// TwinCAT 3 PLC project MobilePlatform
// ProgramVersion: 3.1.4022.7
// libraries:
//   Tc2_EtherCAT, * (Beckhoff Automation GmbH)
//   Tc2_Math, * (Beckhoff Automation GmbH)
//   Tc2_MC2, * (Beckhoff Automation GmbH)
//   Tc2_Standard, * (Beckhoff Automation GmbH)
//   Tc2_SUPS, * (Beckhoff Automation GmbH)
//   Tc2_System, * (Beckhoff Automation GmbH)
//   Tc2_TcpIp, * (Beckhoff Automation GmbH)
//   Tc2_Utilities, * (Beckhoff Automation GmbH)
//   Tc3_Module, * (Beckhoff Automation GmbH)
// project tree:
//   DUTs/ ButtonType.TcDUT, ByteDword.TcDUT, ByteReal.TcDUT, ControlerState.TcDUT, DirPlatform.TcDUT, E_ClientServerSteps.TcDUT, E_CONTROL_STATES.TcDUT, InternalState.TcDUT, JoystickCalibState.TcDUT, JoystickState.TcDUT, LEDtype.TcDUT, RealDword.TcDUT, ST_Calibration_Parameters.TcDUT, ST_FrameFifoEntry.TcDUT
//   GVLs/ ControlGVL.TcGVL, JoystickGVL.TcGVL, MOTORS.TcGVL, SafetyGVL.TcGVL, SensorsGVL.TcGVL
//   POUs/Joystick/FBs/ AXISdriver.TcPOU, BUTTONdriver.TcPOU, CalibrationFB.TcPOU, LEDdriver.TcPOU
//   POUs/Joystick/ JoystickMain.TcPOU
//   POUs/Motors/FBs/ FB_RESET_MOTORS.TcPOU, FB_RUN_MOTOR.TcPOU
//   POUs/Motors/ MAIN.TcPOU
//   POUs/Sensors/ SensorsMain.TcPOU
//   / Task1.TcTTO, Task3.TcTTO, Task_2.TcTTO
// real-time tasks:
//   TASK Task1: cycle T#50us, priority 6, ADS port 350
//   TASK Task3: cycle T#10ms, priority 12, ADS port 360
//   TASK Task 2: cycle T#1ms, priority 7, ADS port 351
// motion (NC):
//   TASK NC-Task 1 SAF: cycle T#500us, priority 8, ADS port 501
//   TASK NC-Task 1 SVB: cycle T#10ms, priority 14, ADS port 511
//   AXIS Wheel_Back_Left (id 1)
//     General: UnitName=°
//     Dynamic: Acceleration=30537, Deceleration=30537, Jerk=91611
//     Velo: RefSearch=203.58, RefSync=203.58, SlowManual=1017.9, FastManual=6107.4, Fast=20358, Maximum=20358
//     OtherSettings: AllowMotionCmdToSlave=true
//     encoder EncType=19
//       EncPara: ScaleFactorNumerator=360, ScaleFactorDenominator=1048576, MaxCount=#xffffffff
//     drive DrvType=16
//       DrvPara: MaxCount=#xffffffff, DriveControlDWord=#x00020000
//         Analog: VeloReferenz=22393.8, VeloScale=32, ScaleFactorActTorque=0.1
//         TimeComp: TaskDelayCycles=1
//     controller CtrType=1
//       CtrPara: PriorControlFactor=1
//         PosDiffControl: Enable=false
//         Observer: BandWidth=20
//   AXIS Wheel_Back_Right (id 2)
//     General: UnitName=°
//     Dynamic: Acceleration=30537, Deceleration=30537, Jerk=91611
//     Velo: RefSearch=203.58, RefSync=203.58, SlowManual=1017.9, FastManual=6107.4, Fast=20358, Maximum=20358
//     OtherSettings: AllowMotionCmdToSlave=true
//     encoder EncType=19
//       EncPara: ScaleFactorNumerator=360, ScaleFactorDenominator=1048576, MaxCount=#xffffffff
//     drive DrvType=16
//       DrvPara: MaxCount=#xffffffff, DriveControlDWord=#x00020000
//         Analog: VeloReferenz=22393.8, VeloScale=32, ScaleFactorActTorque=0.1
//         TimeComp: TaskDelayCycles=1
//     controller CtrType=1
//       CtrPara: PriorControlFactor=1
//         PosDiffControl: Enable=false
//         Observer: BandWidth=20
//   AXIS Wheel_Front_Left (id 3)
//     General: UnitName=°
//     Dynamic: Acceleration=30537, Deceleration=30537, Jerk=91611
//     Velo: RefSearch=203.58, RefSync=203.58, SlowManual=1017.9, FastManual=6107.4, Fast=20358, Maximum=20358
//     OtherSettings: AllowMotionCmdToSlave=true
//     encoder EncType=19
//       EncPara: ScaleFactorNumerator=360, ScaleFactorDenominator=1048576, MaxCount=#xffffffff
//     drive DrvType=16
//       DrvPara: MaxCount=#xffffffff, DriveControlDWord=#x00020000
//         Analog: VeloReferenz=22393.8, VeloScale=32, ScaleFactorActTorque=0.1
//         TimeComp: TaskDelayCycles=1
//     controller CtrType=1
//       CtrPara: PriorControlFactor=1
//         PosDiffControl: Enable=false
//         Observer: BandWidth=20
//   AXIS Wheel_Front_Right (id 4)
//     General: UnitName=°
//     Dynamic: Acceleration=30537, Deceleration=30537, Jerk=91611
//     Velo: RefSearch=203.58, RefSync=203.58, SlowManual=1017.9, FastManual=6107.4, Fast=20358, Maximum=20358
//     OtherSettings: AllowMotionCmdToSlave=true
//     encoder EncType=19
//       EncPara: ScaleFactorNumerator=360, ScaleFactorDenominator=1048576, MaxCount=#xffffffff
//     drive DrvType=16
//       DrvPara: MaxCount=#xffffffff, DriveControlDWord=#x00020000
//         Analog: VeloReferenz=22393.8, VeloScale=32, ScaleFactorActTorque=0.1
//         TimeComp: TaskDelayCycles=1
//     controller CtrType=1
//       CtrPara: PriorControlFactor=1
//         PosDiffControl: Enable=false
//         Observer: BandWidth=20
// I/O:
//   DEVICE Device 1 (EtherCAT), AmsNetId 5.51.149.114.2.1
//     Term 1 (EK1200) [EK1200-5000 EtherCAT Power supply (2A E-Bus)]
//       Term 2 (EL3008) [EL3008 8Ch. Ana. Input +/-10V]
//       Term 3 (EL1259) [EL1259 8Ch. Dig Input 24V/8Ch. Dig. Output 24V with Multi-Time-Stamp]
//       Term 4 (EL7211-9014) [EL7211-9014 1Ch. MDP742 Servo motor output stage with OCT (50V, 4.5A RMS) and STO input]
//       Term 5 (EL7211-9014) [EL7211-9014 1Ch. MDP742 Servo motor output stage with OCT (50V, 4.5A RMS) and STO input]
//       Term 6 (EL2904) [EL2904, 4 Ch. Safety Output 24V, 0.5A, TwinSAFE]
//         modules: Module 1 (FSOES), Module 2 (DO)
//       Term 7 (EL7211-9014) [EL7211-9014 1Ch. MDP742 Servo motor output stage with OCT (50V, 4.5A RMS) and STO input]
//       Term 8 (EL7211-9014) [EL7211-9014 1Ch. MDP742 Servo motor output stage with OCT (50V, 4.5A RMS) and STO input]
//       Term 9 (EL1904) [EL1904, 4 Ch. Safety Input 24V, TwinSAFE]
//         modules: Module 1 (FSOES)
//       Term 10 (EL6900) [EL6900, TwinSAFE PLC]
//       Term 11 (EL6070) [EL6070 1Ch. Licensing-Terminal]
//       Term 12 (EL9011) [EL9011 End Terminal]
// variable links:
//   Device 1 (EtherCAT) <-> Device 1 (EtherCAT)/Term 1 (EK1200)/Term 10 (EL6900)
//     Term 1 (EK1200)/Term 6 (EL2904)/Module 1 (FSOES)/RxPDO/FSOE <-> ConnectionInputs/Message_2 TxPDO
//     Term 1 (EK1200)/Term 9 (EL1904)/Module 1 (FSOES)/RxPDO/FSOE <-> ConnectionInputs/Message_3 TxPDO
//   Device 1 (EtherCAT) <-> Device 1 (EtherCAT)/Term 1 (EK1200)/Term 6 (EL2904)
//     Term 1 (EK1200)/Term 10 (EL6900)/ConnectionOutputs/Message_2 RxPDO <-> Module 1 (FSOES)/TxPDO/FSOE
//   Device 1 (EtherCAT) <-> Device 1 (EtherCAT)/Term 1 (EK1200)/Term 9 (EL1904)
//     Term 1 (EK1200)/Term 10 (EL6900)/ConnectionOutputs/Message_3 RxPDO <-> Module 1 (FSOES)/TxPDO/FSOE
//   NC-Task 1 SAF/Axes/Wheel_Back_Left <-> Device 1 (EtherCAT)/Term 1 (EK1200)/Term 4 (EL7211-9014)
//     Drive/Inputs/In/nDcOutputTime <-> InfoData/DcOutputShift
//     Drive/Inputs/In/nState1 <-> DRV Statusword/Statusword
//     Drive/Inputs/In/nState2 <-> DRV Statusword/Statusword @bit 8
//     Drive/Inputs/In/nState4 @bit 1 <-> WcState/InputToggle
//     Drive/Inputs/In/nState4 <-> WcState/WcState
//     Drive/Outputs/Out/nCtrl1 <-> DRV Controlword/Controlword
//     Drive/Outputs/Out/nCtrl2 <-> DRV Controlword/Controlword @bit 8
//     Drive/Outputs/Out/nDataOut2 <-> DRV Target velocity/Target velocity
//     Enc/Inputs/In/nDataIn1 <-> FB Position/Position
//     Enc/Inputs/In/nDcInputTime <-> InfoData/DcInputShift
//     Enc/Inputs/In/nState4 @bit 1 <-> WcState/InputToggle
//     Enc/Inputs/In/nState4 <-> WcState/WcState
//   NC-Task 1 SAF/Axes/Wheel_Back_Right <-> Device 1 (EtherCAT)/Term 1 (EK1200)/Term 5 (EL7211-9014)
//     Drive/Inputs/In/nDcOutputTime <-> InfoData/DcOutputShift
//     Drive/Inputs/In/nState1 <-> DRV Statusword/Statusword
//     Drive/Inputs/In/nState2 <-> DRV Statusword/Statusword @bit 8
//     Drive/Inputs/In/nState4 @bit 1 <-> WcState/InputToggle
//     Drive/Inputs/In/nState4 <-> WcState/WcState
//     Drive/Outputs/Out/nCtrl1 <-> DRV Controlword/Controlword
//     Drive/Outputs/Out/nCtrl2 <-> DRV Controlword/Controlword @bit 8
//     Drive/Outputs/Out/nDataOut2 <-> DRV Target velocity/Target velocity
//     Enc/Inputs/In/nDataIn1 <-> FB Position/Position
//     Enc/Inputs/In/nDcInputTime <-> InfoData/DcInputShift
//     Enc/Inputs/In/nState4 @bit 1 <-> WcState/InputToggle
//     Enc/Inputs/In/nState4 <-> WcState/WcState
//   NC-Task 1 SAF/Axes/Wheel_Front_Left <-> Device 1 (EtherCAT)/Term 1 (EK1200)/Term 7 (EL7211-9014)
//     Drive/Inputs/In/nDcOutputTime <-> InfoData/DcOutputShift
//     Drive/Inputs/In/nState1 <-> DRV Statusword/Statusword
//     Drive/Inputs/In/nState2 <-> DRV Statusword/Statusword @bit 8
//     Drive/Inputs/In/nState4 @bit 1 <-> WcState/InputToggle
//     Drive/Inputs/In/nState4 <-> WcState/WcState
//     Drive/Outputs/Out/nCtrl1 <-> DRV Controlword/Controlword
//     Drive/Outputs/Out/nCtrl2 <-> DRV Controlword/Controlword @bit 8
//     Drive/Outputs/Out/nDataOut2 <-> DRV Target velocity/Target velocity
//     Enc/Inputs/In/nDataIn1 <-> FB Position/Position
//     Enc/Inputs/In/nDcInputTime <-> InfoData/DcInputShift
//     Enc/Inputs/In/nState4 @bit 1 <-> WcState/InputToggle
//     Enc/Inputs/In/nState4 <-> WcState/WcState
//   NC-Task 1 SAF/Axes/Wheel_Front_Right <-> Device 1 (EtherCAT)/Term 1 (EK1200)/Term 8 (EL7211-9014)
//     Drive/Inputs/In/nDcOutputTime <-> InfoData/DcOutputShift
//     Drive/Inputs/In/nState1 <-> DRV Statusword/Statusword
//     Drive/Inputs/In/nState2 <-> DRV Statusword/Statusword @bit 8
//     Drive/Inputs/In/nState4 @bit 1 <-> WcState/InputToggle
//     Drive/Inputs/In/nState4 <-> WcState/WcState
//     Drive/Outputs/Out/nCtrl1 <-> DRV Controlword/Controlword
//     Drive/Outputs/Out/nCtrl2 <-> DRV Controlword/Controlword @bit 8
//     Drive/Outputs/Out/nDataOut2 <-> DRV Target velocity/Target velocity
//     Enc/Inputs/In/nDataIn1 <-> FB Position/Position
//     Enc/Inputs/In/nDcInputTime <-> InfoData/DcInputShift
//     Enc/Inputs/In/nState4 @bit 1 <-> WcState/InputToggle
//     Enc/Inputs/In/nState4 <-> WcState/WcState
//   MobilePlatform/MobilePlatform Instance <-> Device 1 (EtherCAT)/Term 1 (EK1200)/Term 10 (EL6900)
//     Task1 Inputs/SafetyGVL.ComErr <-> StandardInputs/Standard Out Var 4
//     Task1 Inputs/SafetyGVL.EStop <-> StandardInputs/Standard Out Var 5
//     Task1 Outputs/SafetyGVL.ErrAck <-> StandardOutputs/Standard In Var 1
//   MobilePlatform/MobilePlatform Instance <-> Device 1 (EtherCAT)/Term 1 (EK1200)/Term 2 (EL3008)
//     Task3 Inputs/JoystickMain.axDr.xRaw <-> AI Standard Channel 1/Value
//     Task3 Inputs/JoystickMain.axDr.yRaw <-> AI Standard Channel 2/Value
//     Task3 Inputs/JoystickMain.axDr.zRaw <-> AI Standard Channel 3/Value
//     Task3 Inputs/JoystickMain.calFB.axDr.xRaw <-> AI Standard Channel 1/Value
//     Task3 Inputs/JoystickMain.calFB.axDr.yRaw <-> AI Standard Channel 2/Value
//     Task3 Inputs/JoystickMain.calFB.axDr.zRaw <-> AI Standard Channel 3/Value
//   MobilePlatform/MobilePlatform Instance <-> Device 1 (EtherCAT)/Term 1 (EK1200)/Term 3 (EL1259)
//     Task3 Inputs/JoystickMain.btDR.ch1 <-> MTI Inputs 10x Channel 1/Status/Input state
//     Task3 Inputs/JoystickMain.btDR.ch8 <-> MTI Inputs 10x Channel 8/Status/Input state
//     Task3 Outputs/JoystickMain.ldDr1.ch1 <-> MTO Outputs 10x Channel 1/Ctrl/Manual output state
//     Task3 Outputs/JoystickMain.ldDr3.ch3 <-> MTO Outputs 10x Channel 3/Ctrl/Manual output state
//     Task3 Outputs/JoystickMain.ldDr1.ch1mode <-> MTO Outputs 10x Channel 1/Ctrl/Enable manual operation
//     Task3 Outputs/JoystickMain.ldDr3.ch3mode <-> MTO Outputs 10x Channel 3/Ctrl/Enable manual operation
//     Task_2 Inputs/SensorsMain.sensor1_UO1 <-> MTI Inputs 10x Channel 5/Status/Input state
//     Task_2 Inputs/SensorsMain.sensor1_UO2 <-> MTI Inputs 10x Channel 6/Status/Input state
//     Task_2 Inputs/SensorsMain.sensor1_UO3 <-> MTI Inputs 10x Channel 4/Status/Input state
//     Task_2 Inputs/SensorsMain.sensor2_UO1 <-> MTI Inputs 10x Channel 2/Status/Input state
//     Task_2 Inputs/SensorsMain.sensor2_UO2 <-> MTI Inputs 10x Channel 3/Status/Input state
//     Task_2 Inputs/SensorsMain.sensor2_UO3 <-> MTI Inputs 10x Channel 7/Status/Input state
//     Task_2 Outputs/SensorsMain.en_sensor1_D <-> MTO Outputs 10x Channel 6/Ctrl/Enable manual operation
//     Task_2 Outputs/SensorsMain.en_sensor2_D <-> MTO Outputs 10x Channel 5/Ctrl/Enable manual operation
//     Task_2 Outputs/SensorsMain.en_sensor1_E <-> MTO Outputs 10x Channel 7/Ctrl/Enable manual operation
//     Task_2 Outputs/SensorsMain.en_sensor2_E <-> MTO Outputs 10x Channel 4/Ctrl/Enable manual operation
//     Task_2 Outputs/SensorsMain.en_sensor1_F <-> MTO Outputs 10x Channel 8/Ctrl/Enable manual operation
//     Task_2 Outputs/SensorsMain.en_sensor2_F <-> MTO Outputs 10x Channel 2/Ctrl/Enable manual operation
//     Task_2 Outputs/SensorsMain.sensor1_D <-> MTO Outputs 10x Channel 6/Ctrl/Manual output state
//     Task_2 Outputs/SensorsMain.sensor2_D <-> MTO Outputs 10x Channel 5/Ctrl/Manual output state
//     Task_2 Outputs/SensorsMain.sensor1_E <-> MTO Outputs 10x Channel 7/Ctrl/Manual output state
//     Task_2 Outputs/SensorsMain.sensor2_E <-> MTO Outputs 10x Channel 4/Ctrl/Manual output state
//     Task_2 Outputs/SensorsMain.sensor1_F <-> MTO Outputs 10x Channel 8/Ctrl/Manual output state
//     Task_2 Outputs/SensorsMain.sensor2_F <-> MTO Outputs 10x Channel 2/Ctrl/Manual output state
//   MobilePlatform/MobilePlatform Instance <-> NC-Task 1 SAF/Axes/Wheel_Back_Left
//     Task1 Inputs/MOTORS.fbAxisRef_BL.NcToPlc <-> Outputs/ToPlc
//     Task1 Outputs/MOTORS.fbAxisRef_BL.PlcToNc <-> Inputs/FromPlc
//   MobilePlatform/MobilePlatform Instance <-> NC-Task 1 SAF/Axes/Wheel_Back_Right
//     Task1 Inputs/MOTORS.fbAxisRef_BR.NcToPlc <-> Outputs/ToPlc
//     Task1 Outputs/MOTORS.fbAxisRef_BR.PlcToNc <-> Inputs/FromPlc
//   MobilePlatform/MobilePlatform Instance <-> NC-Task 1 SAF/Axes/Wheel_Front_Left
//     Task1 Inputs/MOTORS.fbAxisRef_FL.NcToPlc <-> Outputs/ToPlc
//     Task1 Outputs/MOTORS.fbAxisRef_FL.PlcToNc <-> Inputs/FromPlc
//   MobilePlatform/MobilePlatform Instance <-> NC-Task 1 SAF/Axes/Wheel_Front_Right
//     Task1 Inputs/MOTORS.fbAxisRef_FR.NcToPlc <-> Outputs/ToPlc
//     Task1 Outputs/MOTORS.fbAxisRef_FR.PlcToNc <-> Inputs/FromPlc

CONFIGURATION MobilePlatform
    RESOURCE PLC ON TwinCAT3
        TASK Task1(INTERVAL := T#50us, PRIORITY := 6);
        TASK Task3(INTERVAL := T#10ms, PRIORITY := 12);
        TASK Task_2(INTERVAL := T#1ms, PRIORITY := 7);
        PROGRAM MAIN WITH Task1 : MAIN;
        PROGRAM JoystickMain WITH Task3 : JoystickMain;
        PROGRAM SensorsMain WITH Task_2 : SensorsMain;
    END_RESOURCE
END_CONFIGURATION

// ---- DUTs/ButtonType.TcDUT
{attribute 'qualified_only'}
//{attribute 'strict'}
TYPE ButtonType :
(
	notPressed := 0,
	pressed := 1,
	hold2s := 2,
	hold5s := 5
);
END_TYPE

// ---- DUTs/ByteDword.TcDUT
TYPE ByteDword :
UNION
	dValue : DWORD;    // Needs 4 Bytes in memory
    abValue:  ARRAY [1..4] OF BYTE;
END_UNION
END_TYPE

// ---- DUTs/ByteReal.TcDUT
TYPE ByteReal :
UNION
	rValue : REAL;    // Needs 4 Bytes in memory
    abValue:  ARRAY [1..4] OF BYTE;
END_UNION
END_TYPE

// ---- DUTs/ControlerState.TcDUT
{attribute 'qualified_only'}
{attribute 'strict'}
TYPE ControlerState :
(
	UDPcontrol := 0,
	LocalOverride := 1,
	Blocked := 2
);
END_TYPE

// ---- DUTs/DirPlatform.TcDUT
{attribute 'qualified_only'}
{attribute 'strict'}
TYPE DirPlatform :
(
	
	PLUS_X := 0,
	PLUS_X_MINUS_Y := 1,
	MINUS_Y := 2,
	MINUS_X_MINUS_Y := 3,
	MINUS_X := 4,
	MINUS_X_PLUS_Y := 5,
	PLUS_Y := 6,
	PLUS_X_PLUS_Y := 7
);
END_TYPE

// ---- DUTs/E_ClientServerSteps.TcDUT
TYPE E_ClientServerSteps :
(
	eUDP_STATE_IDLE		:= 0,
	eUDP_STATE_CREATE_START,
	eUDP_STATE_CREATE_WAIT,
	eUDP_STATE_SEND_START,
	eUDP_STATE_SEND_WAIT,
	eUDP_STATE_RECEIVE_START,
	eUDP_STATE_RECEIVE_WAIT,
	eUDP_STATE_CLOSE_START,
	eUDP_STATE_CLOSE_WAIT,
	eUDP_STATE_ERROR
);
END_TYPE

// ---- DUTs/E_CONTROL_STATES.TcDUT
TYPE E_CONTROL_STATES :
(
	eControlState_Preinit := 100,
	eControlState_Init := 110,
	eControlState_Hold := 120,
	eControlState_Move := 130,
	eControlState_Move_Omni := 140,
	eControlState_Move_Omni_Rot := 150
	);
END_TYPE

// ---- DUTs/InternalState.TcDUT
{attribute 'qualified_only'}
{attribute 'strict'}
TYPE InternalState :
(
	passive := 0,
	override := 1,
	udpOnly := 2
);
END_TYPE

// ---- DUTs/JoystickCalibState.TcDUT
{attribute 'qualified_only'}
{attribute 'strict'}
TYPE JoystickCalibState :
(
	CalibMinMax := 0,
	CalibDeadband := 1,
	CalibOver := 2,
	CalibStart := 3
);
END_TYPE

// ---- DUTs/JoystickState.TcDUT
{attribute 'qualified_only'}
{attribute 'strict'}
TYPE JoystickState :
(
	NoCalib := 0,
	Operational := 1,
	Calib := 2
);
END_TYPE

// ---- DUTs/LEDtype.TcDUT
{attribute 'qualified_only'}
{attribute 'strict'}
TYPE LEDtype :
(
	OFF := 0,
	ON := 1,
	Pulse := 2,
	BlinkOnce := 3,
	BlinkContinious := 4
);
END_TYPE

// ---- DUTs/RealDword.TcDUT
TYPE RealDword :
UNION
	rValue : REAL;
	dValue : DWORD;
END_UNION
END_TYPE

// ---- DUTs/ST_Calibration_Parameters.TcDUT
TYPE ST_Calibration_Parameters :
STRUCT
	maximums : ARRAY [1..3] OF INT;
	minimums : ARRAY [1..3] OF INT;
	deadband : ARRAY [1..3] OF INT;
	zero     : ARRAY [1..3] OF INT;
	
	timeOfCalib : DATE_AND_TIME;
	
	calibrated : BOOL := FALSE;
END_STRUCT
END_TYPE

// ---- DUTs/ST_FrameFifoEntry.TcDUT
TYPE ST_FrameFifoEntry :
STRUCT
	stRemoteAddr 	: ST_SockAddr;(* Remote address. String containing an (Ipv4) Internet Protocol dotted address and port number. *)
	sMessage		: ARRAY [0..100] OF BYTE;	(* UDP packet data *)
END_STRUCT
END_TYPE

// ---- GVLs/ControlGVL.TcGVL
{attribute 'qualified_only'}
VAR_GLOBAL


	
	status : DWORD := 0; //status Bit0 - EStop Active, Bit1 - Manual override, Bit2 - JoystickUdp only, Bit3 - 9 Joystick states
	//all values in deg or deg/s
	vel_BL : LREAL := 0.0;
	vel_BR : LREAL := 0.0;
	vel_FL : LREAL := 0.0;
	vel_FR : LREAL := 0.0;
	
	pos_BL : LREAL := 0.0;
	pos_BR : LREAL := 0.0;
	pos_FL : LREAL := 0.0;
	pos_FR : LREAL := 0.0;
	
	leftRight : LREAL := 0; // left-right command 
	forwardReverse : LREAL := 0; // forward-reverse comand
	rotLeftRight : LREAL := 0;
	
	TimeStamp : LREAL := 0.0;
	
	vel_robot : ARRAY [1..3] OF LREAL := [0,0,0]; //commands platform velocity x-y-th + timestamp	from ROS
	robot_odom : ARRAY [1..6] OF LREAL := [0,0,0,0,0,0]; //acctual position and velocity robot order pos-vel x-y-th
	
	
	currentVelMax : LREAL :=0;
	currentThVelMax : LREAL :=0;
END_VAR

// ---- GVLs/JoystickGVL.TcGVL
{attribute 'qualified_only'}
VAR_GLOBAL
	state : JoystickState := JoystickState.NoCalib;
	xConst : LREAL := -0.3; //x y z max speeds
	yConst : LREAL := 0.2;
	zConst : LREAL := 0.4;
	
	xSpeed : LREAL := 0.0;
	ySpeed : LREAL := 0.0;
	zSpeed : LREAL := 0.0;
	
	speedScale : LREAL := 1.0;
	
	intState : InternalState := InternalState.passive;
	
	lastUpdate : BOOL := FALSE;
	lastExec : BOOL := FALSE;
END_VAR

VAR_GLOBAL PERSISTENT
	calibration : ST_Calibration_Parameters;
END_VAR

// ---- GVLs/MOTORS.TcGVL
{attribute 'qualified_only'}

VAR_GLOBAL
	
    // Axis reference 
    fbAxisRef_BL:				AXIS_REF;
	fbAxisRef_BR:				AXIS_REF;
	fbAxisRef_FL:				AXIS_REF;
	fbAxisRef_FR:				AXIS_REF;
	// Motors' Power
	fbPOWER_BL : 				MC_Power;
    fbPOWER_BR : 				MC_Power;	
    fbPOWER_FL : 				MC_Power;
    fbPOWER_FR : 				MC_Power;		
	// Reset Motors
	fbRESET_BL : 				MC_Reset;
	fbRESET_BR : 				MC_Reset;
	// Stop Motors
	fbSTOP_BL :	 				MC_Stop;
	fbSTOP_BR :	 				MC_Stop;
	// Velocity Controllers 
	fbVELOCITY_BL : 			MC_MoveVelocity;
	fbVELOCITY_BR : 			MC_MoveVelocity;
	fbVELOCITY_FL : 			MC_MoveVelocity;
	fbVELOCITY_FR : 			MC_MoveVelocity;
	// Move absolute - it will move the axis to an absolute position 
	fbMOVEABSOLUTE_LB : 		MC_MoveAbsolute;
	fbMOVEABSOLUTE_RB : 		MC_MoveAbsolute;
	// Set position if mode relative
	fbSETPOSITION_BL : 			MC_SetPosition;
	fbSETPOSITION_BR : 			MC_SetPosition;
    // Move relative - it will move the axis to a relative position
	fbMOVERELATIVE_BL : 		MC_MoveRelative;
	fbMOVERELATIVE_BR : 		MC_MoveRelative;
	// Read actual position of the axis
	fbACTUALPOSITION_BL : 		MC_ReadActualPosition;
	fbACTUALPOSITION_BR : 		MC_ReadActualPosition;
	// Direction enumeration
	fbDirection_BL: 			MC_Direction := MC_Positive_Direction;  // MC_Positive_Direction or MC_Negative_Direction
	fbDirection_BR: 			MC_Direction := MC_Positive_Direction; 
	fbDirection_FL: 			MC_Direction := MC_Positive_Direction;  // MC_Positive_Direction or MC_Negative_Direction
	fbDirection_FR: 			MC_Direction := MC_Positive_Direction; 
	
	// Control Values
	bAxis_Ready : 				BOOL;
	b_Move_Absolut_Aborted : 	BOOL;
	bReset_Done : 				BOOL;
    lrAcc_Axis_1 : 				LREAL;
	lrActual_Position : 		LREAL;
	lrDecel_Axis_1 :			LREAL;
	lrJerk_Axis_1 : 			LREAL;
	lrPosition_Drive_to : 		LREAL;
	lrVelocity_Move_Ab_Axis: 	LREAL;	
	
	//External set point generators enable
	MC_ExtSetPointGenEnableBL : MC_ExtSetPointGenEnable;
	MC_ExtSetPointGenEnableBR : MC_ExtSetPointGenEnable;
	MC_ExtSetPointGenEnableFL : MC_ExtSetPointGenEnable;
	MC_ExtSetPointGenEnableFR : MC_ExtSetPointGenEnable;
	
	//External set point generators disable
	MC_ExtSetPointGenDisableBL : MC_ExtSetPointGenDisable;
	MC_ExtSetPointGenDisableBR : MC_ExtSetPointGenDisable;
	MC_ExtSetPointGenDisableFL : MC_ExtSetPointGenDisable;
	MC_ExtSetPointGenDisableFR : MC_ExtSetPointGenDisable;


	

END_VAR

// ---- GVLs/SafetyGVL.TcGVL
{attribute 'qualified_only'}
VAR_GLOBAL
	ErrAck AT %Q* : BOOL;
	ComErr AT %I* : BOOL;
	EStop AT %I* : BOOL;
END_VAR

// ---- GVLs/SensorsGVL.TcGVL
{attribute 'qualified_only'}
VAR_GLOBAL

	
	platformDir : INT := 0;

END_VAR

// ---- POUs/Motors/MAIN.TcPOU
PROGRAM MAIN
VAR
	

	tmr1 : TON;
	tmr1val : BOOL := FALSE;
	
	estopActive : BOOL := FALSE;
	
	reset1 : FB_RESET_MOTORS;
	
	Enabled : BOOL := TRUE;
	
	fbRunMotor : FB_RUN_MOTOR;
	//leddriver : LEDdriver;
END_VAR

IF SafetyGVL.ComErr = TRUE THEN
	//Safety needs to be reset - reset safety
	SafetyGVL.ErrAck := TRUE;
	tmr1val := TRUE;
END_IF

IF SafetyGVL.EStop = FALSE THEN
		//EStop was activated
		estopActive := TRUE;
		ControlGVL.status := ControlGVL.status OR 2#00000000000000000000000000000001;
END_IF

tmr1(IN := tmr1val, PT := T#1S);

IF (estopActive = TRUE) AND (SafetyGVL.EStop = TRUE) THEN
	//EStop over - reset motor drivers
	reset1();
	IF reset1.EstopOut = FALSE THEN
		ControlGVL.status := ControlGVL.status AND 2#11111111111111111111111111111110;
		estopActive := FALSE;
	END_IF
END_IF

IF tmr1.Q = TRUE THEN
	
	//Safety online - run program
	SafetyGVL.ErrAck := FALSE;
	fbRunMotor();
	//leddriver(ledBlink := LEDtype.ON, blinkInterval := T#1S, ledChannel := 3);
	
END_IF

END_PROGRAM

// ---- POUs/Motors/FBs/FB_RESET_MOTORS.TcPOU
FUNCTION_BLOCK FB_RESET_MOTORS
VAR_INPUT
END_VAR
VAR_OUTPUT
	EstopOut : BOOL := TRUE;
END_VAR
VAR
	tmr1 : TON;
	
	tmr1val : BOOL := FALSE;
	
	reset1 : MC_Reset;
	reset2 : MC_Reset;
	reset3 : MC_Reset;
	reset4 : MC_Reset;
END_VAR

tmr1(IN := tmr1val, PT :=T#2S);

IF tmr1.Q = FALSE THEN
	
	reset1(Axis := MOTORS.fbAxisRef_BL, Execute := TRUE);
	reset2(Axis := MOTORS.fbAxisRef_BR, Execute := TRUE);
	reset3(Axis := MOTORS.fbAxisRef_FR, Execute := TRUE);
	reset4(Axis := MOTORS.fbAxisRef_FL, Execute := TRUE);
	tmr1val := TRUE;
	EstopOut := TRUE;
	
	//disable use of external set point generator
	MOTORS.MC_ExtSetPointGenDisableBL(Axis:=MOTORS.fbAxisRef_BL,
		Execute := TRUE);
	MOTORS.MC_ExtSetPointGenDisableBR(Axis:=MOTORS.fbAxisRef_BR,
		Execute := TRUE);
	MOTORS.MC_ExtSetPointGenDisableFR(Axis:=MOTORS.fbAxisRef_FR,
		Execute := TRUE);
	MOTORS.MC_ExtSetPointGenDisableFL(Axis:=MOTORS.fbAxisRef_FL,
		Execute := TRUE);
			
	//reset enable
	MOTORS.MC_ExtSetPointGenEnableBL(Axis:=MOTORS.fbAxisRef_BL,
		Execute:=FALSE);
	MOTORS.MC_ExtSetPointGenEnableBR(Axis:=MOTORS.fbAxisRef_BR,
		Execute:=FALSE);
	MOTORS.MC_ExtSetPointGenEnableFL(Axis:=MOTORS.fbAxisRef_FL,
		Execute:=FALSE);
	MOTORS.MC_ExtSetPointGenEnableFR(Axis:=MOTORS.fbAxisRef_FR,
		Execute:=FALSE);
	
	
END_IF

IF tmr1.Q = TRUE THEN
	
	reset1(Axis := MOTORS.fbAxisRef_BL, Execute := FALSE);
	reset2(Axis := MOTORS.fbAxisRef_BR, Execute := FALSE);
	reset3(Axis := MOTORS.fbAxisRef_FR, Execute := FALSE);
	reset4(Axis := MOTORS.fbAxisRef_FL, Execute := FALSE);
	tmr1val := FALSE;
	EstopOut := FALSE;
	
	
		
		//Enable use of external set point generator
	MOTORS.MC_ExtSetPointGenEnableBL(Axis:=MOTORS.fbAxisRef_BL,
		Execute:=TRUE,
		Position := 0,
		PositionType:=POSITIONTYPE_ABSOLUTE);
		
	MOTORS.MC_ExtSetPointGenEnableBR(Axis:=MOTORS.fbAxisRef_BR,
		Execute:=TRUE,
		Position := 0,
		PositionType:=POSITIONTYPE_ABSOLUTE);
			
	MOTORS.MC_ExtSetPointGenEnableFL(Axis:=MOTORS.fbAxisRef_FL,
		Execute:=TRUE,
		Position := 0,
		PositionType:=POSITIONTYPE_ABSOLUTE);
			
	MOTORS.MC_ExtSetPointGenEnableFR(Axis:=MOTORS.fbAxisRef_FR,
		Execute:=TRUE,
		Position := 0,
		PositionType:=POSITIONTYPE_ABSOLUTE);
			
	//reset disable external setpoint
	MOTORS.MC_ExtSetPointGenDisableBL(Axis:=MOTORS.fbAxisRef_BL,
		Execute := FALSE);
	MOTORS.MC_ExtSetPointGenDisableBR(Axis:=MOTORS.fbAxisRef_BR,
		Execute := FALSE);	
	MOTORS.MC_ExtSetPointGenDisableFR(Axis:=MOTORS.fbAxisRef_FR,
		Execute := FALSE);	
	MOTORS.MC_ExtSetPointGenDisableFL(Axis:=MOTORS.fbAxisRef_FL,
		Execute := FALSE);
END_IF

END_FUNCTION_BLOCK

// ---- POUs/Motors/FBs/FB_RUN_MOTOR.TcPOU
FUNCTION_BLOCK FB_RUN_MOTOR

VAR
	fbTMR : TON;
    Count : INT := 0;
    
    EnableMoveMotor : BOOL := FALSE;	

	Enabled: BOOL := TRUE;
	Error: BOOL := FALSE;
	ErrorState: BOOL := FALSE;
	oDone: BOOL := FALSE;
	
	userReset : BOOL := FALSE;
	
	xVelocity: LREAL := 0;
	yVelocity: LREAL := 0;
	thVelocity: LREAL := 0;
	


	
	ControlState: INT := eControlState_Preinit;

	Kf: LREAL := 1.0;
	
	
	v_BL_goal : LREAL := 0; // back left motor velocity goal
	v_BR_goal : LREAL := 0; // back right motor velocity goal
	v_FL_goal : LREAL := 0; // front left motor velocity goal
	v_FR_goal : LREAL := 0; // front right motor velocity goal
	
	p_BL : LREAL := 0; // back left motor position
	p_BR : LREAL := 0; // back right motor position
	p_FL : LREAL := 0; // front left motor position
	p_FR : LREAL := 0; // front right motor position
	
	
	v_BL : LREAL := 0; // back left motor velocity 
	v_BR : LREAL := 0; // back right motor velocity
	v_FL : LREAL := 0; // front left motor velocity
	v_FR : LREAL := 0; // front right motor velocity
	
	a_BL : LREAL := 0; // back left motor acceleration
	a_BR : LREAL := 0; // back right motor acceleration
	a_FL : LREAL := 0; // front lefa motor acceleration
	a_FR : LREAL := 0; // front right motor acceleration
	

	CCW : LREAL := 0; // rotation speed command
	
	radioVD : LREAL := 0; // vd from joystick
	radioTH : LREAL := 0; // Theta from joystick
	
	speedC : LREAL := 1.0;
	
	lastTimeStamp : LREAL := -1;
	
	fbReadActualVelocityBL : MC_ReadActualVelocity;
	fbReadActualVelocityBR : MC_ReadActualVelocity;
	fbReadActualVelocityFL : MC_ReadActualVelocity;
	fbReadActualVelocityFR : MC_ReadActualVelocity;
	
	fbReadActualPositionBL : MC_ReadActualPosition;
	fbReadActualPositionBR : MC_ReadActualPosition;
	fbReadActualPositionFL : MC_ReadActualPosition;
	fbReadActualPositionFR : MC_ReadActualPosition;
	
	x : LREAL := 0.0; //real x position
	y : LREAL := 0.0; //real y position
	th : LREAL := 0.0; //real theta position
	
	xV : LREAL := 0.0; //real x velocity
	yV : LREAL := 0.0; //real y velocity
	thV : LREAL := 0.0; //real theta velocity
	
	w_BL : LREAL := 0.0; //back left motor speed
	w_BR : LREAL := 0.0; //back right motor speed
	w_FL : LREAL := 0.0; //front left motor speed
	w_FR : LREAL := 0.0; //front right motor speed
	
	norm : LREAL;
	normWheels : LREAL;

	
	
END_VAR



VAR CONSTANT
	
//slip values
	ax : LREAL := 1.0; //wheel slip
	ar : LREAL := 1.0; //axis/bearing effect
	az : LREAL := 1.0; //rotational grip
	
	//wheel parameters
	rw : LREAL := 0.075; //wheel radius in m
	a  : LREAL := 0.570; //half distance between wheels in y direction
	b  : LREAL := 0.520; //half distance between wheels in x direction
	
	timeSlice: LREAL := 0.00005;
	
	ACC_MAX : LREAL := 7000000;
	VEL_WHEEL_MAX : LREAL := 18000;
	
	//reductor ratio
	RED : LREAL := 16.0;

END_VAR

CASE ControlState OF
	eControlState_Preinit:
	
		// Power on All Motors
    	IF MOTORS.fbPOWER_BL.Active = FALSE THEN
    		MOTORS.fbPOWER_BL(
    			Axis := MOTORS.fbAxisRef_BL, 
    			Enable := Enabled, 
    			Enable_Positive := Enabled, 
    			Enable_Negative := Enabled,
    			BufferMode := MC_Aborting,
    			Override := 100);	
    	END_IF
		
		IF MOTORS.fbPOWER_BR.Active = FALSE THEN
    		MOTORS.fbPOWER_BR(
    			Axis := MOTORS.fbAxisRef_BR, 
    			Enable := Enabled, 
    			Enable_Positive := Enabled, 
    			Enable_Negative := Enabled,
    			BufferMode := MC_Aborting,
    			Override := 100);	
    	END_IF
		
		// Power on All Motors
    	IF MOTORS.fbPOWER_FL.Active = FALSE THEN
    		MOTORS.fbPOWER_FL(
    			Axis := MOTORS.fbAxisRef_FL, 
    			Enable := Enabled, 
    			Enable_Positive := Enabled, 
    			Enable_Negative := Enabled,
    			BufferMode := MC_Aborting,
    			Override := 100);	
    	END_IF
		
		IF MOTORS.fbPOWER_FR.Active = FALSE THEN
    		MOTORS.fbPOWER_FR(
    			Axis := MOTORS.fbAxisRef_FR, 
    			Enable := Enabled, 
    			Enable_Positive := Enabled, 
    			Enable_Negative := Enabled,
    			BufferMode := MC_Aborting,
    			Override := 100);	
    	END_IF

		
		fbTMR(IN:=TRUE, PT:=T#1S);
		
		IF fbTMR.Q THEN
			ControlState := eControlState_Move_Omni;
      		fbTMR(IN:=FALSE);
      	END_IF
		
	eControlState_Move_Omni:
		
		//read actual velocity of motors
		fbReadActualVelocityBL(Axis:= MOTORS.fbAxisRef_BL, Enable := TRUE);
		fbReadActualVelocityBR(Axis:= MOTORS.fbAxisRef_BR, Enable := TRUE);
		fbReadActualVelocityFL(Axis:= MOTORS.fbAxisRef_FL, Enable := TRUE);
		fbReadActualVelocityFR(Axis:= MOTORS.fbAxisRef_FR, Enable := TRUE);
		
		ControlGVL.vel_BL := fbReadActualVelocityBL.ActualVelocity/RED;
		ControlGVL.vel_BR := fbReadActualVelocityBR.ActualVelocity/RED;
		ControlGVL.vel_FL := fbReadActualVelocityFL.ActualVelocity/RED;
		ControlGVL.vel_FR := fbReadActualVelocityFR.ActualVelocity/RED;

		
		//read actual position of motors
		fbReadActualPositionBL(Axis:= MOTORS.fbAxisRef_BL, Enable := TRUE);
		fbReadActualPositionBR(Axis:= MOTORS.fbAxisRef_BR, Enable := TRUE);
		fbReadActualPositionFL(Axis:= MOTORS.fbAxisRef_FL, Enable := TRUE);
		fbReadActualPositionFR(Axis:= MOTORS.fbAxisRef_FR, Enable := TRUE);
		
		ControlGVL.pos_BL :=fbReadActualPositionBL.Position;
		ControlGVL.pos_BR :=fbReadActualPositionBR.Position;
		ControlGVL.pos_FL :=fbReadActualPositionFL.Position;
		ControlGVL.pos_FR :=fbReadActualPositionFR.Position;
		
		//compute odometry
		w_BL := DEG_TO_RAD(ControlGVL.vel_BL);
		w_BR := DEG_TO_RAD(ControlGVL.vel_BR);
		w_FL := DEG_TO_RAD(ControlGVL.vel_FL);
		w_FR := DEG_TO_RAD(ControlGVL.vel_FR);
		
		xV :=    (ax*rw*w_FR)/4 - (ax*rw*w_BL)/4 + (ax*rw*w_BR)/4 - (ax*rw*w_FL)/4;
        yV :=    (ar*ax*rw*w_BL)/4 - (ar*ax*rw*w_FR)/4 + (ar*ax*rw*w_BR)/4 - (ar*ax*rw*w_FL)/4;
 		thV := - (ax*az*2*rw*w_FR)/(4*(a + b)) - (ax*az*2*rw*w_BL)/(4*(a + b)) - (ax*az*rw*2*w_BR)/(4*(a + b)) - (ax*az*2*rw*w_FL)/(4*(a + b));
		
		th := th + thV * timeSlice;
		x := x + xV * timeSlice * COS(th) - yV * timeSlice * SIN(th);
		y := y + yV * timeSlice * COS(th) + xV * timeSlice * SIN(th);
		
		//prepare values to be sent to ROS
		ControlGVL.robot_odom[1] := x;
		ControlGVL.robot_odom[2] := y;
		ControlGVL.robot_odom[3] := th;
		ControlGVL.robot_odom[4] := xV;
		ControlGVL.robot_odom[5] := yV;
		ControlGVL.robot_odom[6] := thV;
		
		//ControlGVL.TimeStamp := ControlGVL.vel_robot[4];
		ControlGVL.TimeStamp := ControlGVL.TimeStamp + 1;
		
		IF (ControlGVL.TimeStamp <> lastTimeStamp OR (JoystickGVL.intState = InternalState.override AND JoystickGVL.state = JoystickState.Operational)) OR JoystickGVL.lastUpdate OR JoystickGVL.lastExec THEN	//If the current instruction has not been executed yet, set speed
		
			
			IF JoystickGVL.lastUpdate THEN
				JoystickGVL.lastUpdate := FALSE;
				ControlGVL.forwardReverse := 0.0;
				ControlGVL.leftRight := 0.0;
				ControlGVL.rotLeftRight := 0.0;
				
			ELSIF (JoystickGVL.state = JoystickState.Operational AND JoystickGVL.intState = InternalState.passive) OR JoystickGVL.state = JoystickState.NoCalib THEN
				//ROS control mode
				ControlGVL.forwardReverse := ControlGVL.vel_robot[1];
				ControlGVL.leftRight := ControlGVL.vel_robot[2];
				ControlGVL.rotLeftRight := ControlGVL.vel_robot[3];
				
				
			ELSIF (JoystickGVL.state = JoystickState.Operational AND JoystickGVL.intState = InternalState.override) THEN
				//Joystick control mode
				ControlGVL.forwardReverse := JoystickGVL.xSpeed * JoystickGVL.xConst * JoystickGVL.speedScale;
				ControlGVL.leftRight := JoystickGVL.ySpeed * JoystickGVL.yConst * JoystickGVL.speedScale;
				ControlGVL.rotLeftRight := JoystickGVL.zSpeed * JoystickGVL.zConst * JoystickGVL.speedScale;

			END_IF
		END_IF
		
		xVelocity := ControlGVL.forwardReverse;
		yVelocity := ControlGVL.leftRight;
		thVelocity := ControlGVL.rotLeftRight;
		
		IF (NOT(JoystickGVL.state = JoystickState.Operational AND JoystickGVL.intState = InternalState.override)) THEN
			//ensure that speed is not too high and adjust it if necessary
				IF( SQRT(xVelocity*xVelocity + yVelocity*yVelocity)>ControlGVL.currentVelMax)THEN
					norm := ABS(xVelocity) + ABS(yVelocity);
					xVelocity := xVelocity*ControlGVL.currentVelMax/norm;
					yVelocity := yVelocity*ControlGVL.currentVelMax/norm;
				END_IF
				
				IF (ABS(thVelocity)>ControlGVL.currentThVelMax) THEN
					thVelocity := thVelocity*ControlGVL.currentThVelMax/ABS(thVelocity);
				END_IF
		END_IF
		
		
		
			
		//set last executed time stamp
		lastTimeStamp := ControlGVL.TimeStamp;
			
		
		//compute velocity goal
		//                     x translation                y translation                 rotation
		v_BL_goal := RAD_TO_DEG(- (ax*xVelocity*RED)/rw + (ax*yVelocity*RED)/(ar*rw) - (ax*thVelocity*RED*(a + b))/(2*az*rw));
		v_BR_goal := RAD_TO_DEG(  (ax*xVelocity*RED)/rw + (ax*yVelocity*RED)/(ar*rw) - (ax*thVelocity*RED*(a + b))/(2*az*rw));
		v_FL_goal := RAD_TO_DEG(- (ax*xVelocity*RED)/rw - (ax*yVelocity*RED)/(ar*rw) - (ax*thVelocity*RED*(a + b))/(2*az*rw));
		v_FR_goal := RAD_TO_DEG(  (ax*xVelocity*RED)/rw - (ax*yVelocity*RED)/(ar*rw) - (ax*thVelocity*RED*(a + b))/(2*az*rw));	
		
		//limit maximum speed of the wheels 
		IF((ABS(v_BL_goal)>VEL_WHEEL_MAX) OR (ABS(v_BR_goal)>VEL_WHEEL_MAX) OR (ABS(v_FL_goal)>VEL_WHEEL_MAX) OR (ABS(v_FR_goal)>VEL_WHEEL_MAX)) THEN
			
			normWheels := VEL_WHEEL_MAX/MAX(ABS(v_BL_goal), ABS(v_BR_goal),ABS(v_FL_goal), ABS(v_FR_goal)); 

			v_BL_goal := v_BL_goal*normWheels;
			v_BR_goal := v_BR_goal*normWheels;
			v_FL_goal := v_FL_goal*normWheels;
			v_FR_goal := v_FR_goal*normWheels;
		END_IF
			
		//derivate to get new acceleration
		a_BL := (v_BL_goal - ControlGVL.vel_BL*RED)/timeSlice;
		a_BR := (v_BR_goal - ControlGVL.vel_BR*RED)/timeSlice;
		a_FL := (v_FL_goal -  ControlGVL.vel_FL*RED)/timeSlice;
		a_FR := (v_FR_goal - ControlGVL.vel_FR*RED)/timeSlice;
		
		IF ABS(a_BL) > ACC_MAX THEN
			a_BL := a_BL*ACC_MAX/ABS(a_BL);
		END_IF
		IF ABS(a_BR) > ACC_MAX THEN
			a_BR := a_BR*ACC_MAX/ABS(a_BR);
		END_IF
		IF ABS(a_FL) > ACC_MAX THEN
			a_FL := a_FL*ACC_MAX/ABS(a_FL);
		END_IF
		IF ABS(a_FR) > ACC_MAX THEN
			a_FR := a_FR*ACC_MAX/ABS(a_FR);
		END_IF

		//integrate to get new velocity
		v_BL := ControlGVL.vel_BL*RED + timeSlice*a_BL;
		v_BR := ControlGVL.vel_BR*RED + timeSlice*a_BR;
		v_FL := ControlGVL.vel_FL*RED + timeSlice*a_FL;
		v_FR := ControlGVL.vel_FR*RED + timeSlice*a_FR;
		
		
		//limit maximum speed of the wheels 
		IF((ABS(v_BL)>VEL_WHEEL_MAX) OR (ABS(v_BR)>VEL_WHEEL_MAX) OR (ABS(v_FL)>VEL_WHEEL_MAX) OR (ABS(v_FR)>VEL_WHEEL_MAX)) THEN
			normWheels := VEL_WHEEL_MAX/MAX(ABS(v_BL), ABS(v_BR),ABS(v_FL), ABS(v_FR)); 

			v_BL := v_BL*normWheels;
			v_BR := v_BR*normWheels;
			v_FL := v_FL*normWheels;
			v_FR := v_FR*normWheels;
			
			a_BL := (v_BL - ControlGVL.vel_BL*RED)/timeSlice;
			a_BR := (v_BR - ControlGVL.vel_BR*RED)/timeSlice;
			a_FL := (v_FL -  ControlGVL.vel_FL*RED)/timeSlice;
			a_FR := (v_FR - ControlGVL.vel_FR*RED)/timeSlice;
		END_IF
		
		//integrate to get new position
		p_BL := ControlGVL.pos_BL + timeSlice*v_BL;
		p_BR := ControlGVL.pos_BR + timeSlice*v_BR;
		p_FL := ControlGVL.pos_FL + timeSlice*v_FL;
		p_FR := ControlGVL.pos_FR + timeSlice*v_FR;
		
		//update values
		MC_ExtSetPointGenFeed(Position := p_BL,
			Velocity := v_BL,
			Acceleration := a_BL,
			Direction := 1,
			Axis := MOTORS.fbAxisRef_BL);
			
		MC_ExtSetPointGenFeed(Position := p_BR,
			Velocity := v_BR,
			Acceleration := a_BR,
			Direction := 1,
			Axis := MOTORS.fbAxisRef_BR);
			
		MC_ExtSetPointGenFeed(Position := p_FL,
			Velocity := v_FL,
			Acceleration := a_FL,
			Direction := 1,
			Axis := MOTORS.fbAxisRef_FL);
			
				
		MC_ExtSetPointGenFeed(Position := p_FR,
			Velocity := v_FR,
			Acceleration := a_FR,
			Direction := 1,
			Axis := MOTORS.fbAxisRef_FR);
			
			
		
END_CASE

END_FUNCTION_BLOCK

// ---- POUs/Joystick/JoystickMain.TcPOU
PROGRAM JoystickMain
VAR
	
	axDr : AXISdriver;
	btDR : BUTTONdriver;
	ldDr1 : LEDdriver;
	ldDr2 : LEDdriver;
	ldDr3 : LEDdriver;
	calFB : CalibrationFB;
	button : ButtonType := ButtonType.notPressed;
	
	prevStateCal : UINT := 0;
	changeState : BOOL := FALSE;
	
	init : BOOL := TRUE;
	initOp : BOOL := TRUE;
	
	WPDfb : WritePersistentData;
	ShtDNfb : FB_S_UPS_CX51x0;
END_VAR

ShtDNfb(sNetID:='', iPLCPort:=0, iUPSPort:=16#588, tTimeout:=DEFAULT_ADS_TIMEOUT, eUpsMode := eSUPS_ImmediateShutdown);
IF NOT ShtDNfb.bPowerFailDetect THEN


	btDr(buttonChannel := 1);
	btDr.getValue(stateOut => button);
	
	WPDfb();
	
	
	CASE JoystickGVL.state OF
		
		JoystickState.NoCalib:
			IF JoystickGVL.calibration.calibrated = TRUE THEN
				JoystickGVL.state := JoystickState.Operational;
				ldDr1(ledChannel := 1, ledBlink := LEDtype.OFF);//zelena
				//ldDr2(ledChannel := 2, ledBlink := LEDtype.OFF);//rumena
				ldDr3(ledChannel := 3, ledBlink := LEDtype.OFF);//rdeca
			ELSE
				ldDr1(ledChannel := 1, ledBlink := LEDtype.OFF);//zelena
				//ldDr2(ledChannel := 2, ledBlink := LEDtype.OFF);//rumena
				IF init THEN
					ldDr3(ledChannel := 3, ledBlink := LEDtype.OFF);//rdeca
					init := FALSE;
				END_IF
				ldDr3(ledChannel := 3, ledBlink := LEDtype.BlinkContinious, blinkInterval := T#0.2S);//rdeca
				IF button = ButtonType.hold5s THEN
					ldDr1(ledChannel := 1, ledBlink := LEDtype.OFF);//zelena
					ldDr2(ledChannel := 2, ledBlink := LEDtype.OFF);//rumena
					ldDr3(ledChannel := 3, ledBlink := LEDtype.OFF);//rdeca
					JoystickGVL.state := JoystickState.Calib;
				END_IF
			END_IF
				
		JoystickState.Calib:
			
			
			calFB(buttonState := button);
			IF calFB.finished THEN
				JoystickGVL.state := JoystickState.Operational;
				JoystickGVL.calibration := calFB.calibrationParams;
				//save here
				WPDfb(START:=0);
				WPDfb(NETID := '', 	PORT:=801, START:=1, TMOUT := T#1S);
				ldDr1(ledChannel := 1, ledBlink := LEDtype.OFF);//zelena
				//ldDr2(ledChannel := 2, ledBlink := LEDtype.OFF);//rumena
				ldDr3(ledChannel := 3, ledBlink := LEDtype.OFF);//rdeca
			END_IF
			IF calFB.calLight THEN
				ldDR3(ledChannel := 3, ledBLink := LEDtype.OFF);
				ldDR3(ledChannel := 3, ledBLink := LEDtype.BlinkOnce);
			END_IF
			IF calFB.stage1 AND NOT (prevStateCal = 1) THEN
				ldDr1(ledChannel := 1, ledBlink := LEDtype.OFF);//zelena
				//ldDr2(ledChannel := 2, ledBlink := LEDtype.OFF);//rumena
				ldDr3(ledChannel := 3, ledBlink := LEDtype.OFF);//rdeca
				ldDr1(ledChannel := 1, ledBlink := LEDtype.BlinkContinious, blinkInterval := T#1S);//rumena
				prevStateCal := 1;
			ELSIF calFB.stage2 AND NOT (prevStateCal = 2) THEN
				ldDr1(ledChannel := 1, ledBlink := LEDtype.OFF);//zelena
				//ldDr2(ledChannel := 2, ledBlink := LEDtype.OFF);//rumena
				ldDr3(ledChannel := 3, ledBlink := LEDtype.OFF);//rdeca
				//ldDr2(ledChannel := 2, ledBlink := LEDtype.BlinkContinious, blinkInterval := T#0.5S);//rumena
				prevStateCal := 2;
			ELSIF calFB.stage3 AND NOT (prevStateCal = 3) THEN
				ldDr1(ledChannel := 1, ledBlink := LEDtype.OFF);//zelena
				//ldDr2(ledChannel := 2, ledBlink := LEDtype.OFF);//rumena
				ldDr3(ledChannel := 3, ledBlink := LEDtype.OFF);//rdeca
				ldDr1(ledChannel := 1, ledBlink := LEDtype.BlinkContinious, blinkInterval := T#0.2S);//rumena
				prevStateCal := 3;
			ELSE
				ldDr1(ledChannel := 1);//zelena
				//ldDr2(ledChannel := 2);//rumena
				ldDr3(ledChannel := 3);//rdeca
			END_IF
			IF  button = ButtonType.hold5s THEN
				JoystickGVL.state := JoystickState.NoCalib;
				ldDr1(ledChannel := 1, ledBlink := LEDtype.OFF);//zelena
				ldDr2(ledChannel := 2, ledBlink := LEDtype.OFF);//rumena
				ldDr3(ledChannel := 3, ledBlink := LEDtype.OFF);//rdeca
				prevStateCal := 0;
				calFB.reset();
				init := TRUE;
			END_IF
		
		JoystickState.Operational:
			
			IF initOp THEN
				initOp := FALSE;
				JoystickGVL.intState := InternalState.passive;
				ControlGVL.status := ControlGVL.status AND 2#11111111111111111111111111111011;
				ldDr3(ledChannel := 3, ledBlink := LEDtype.OFF);
				//ldDr3(ledChannel := 3, ledBlink := LEDtype.ON);
				ldDr1(ledChannel := 1, ledBlink := LEDtype.OFF);//rumena
				ldDr1(ledChannel := 1, ledBlink := LEDtype.ON);//rumena
				//ldDr2(ledChannel := 2, ledBlink := LEDtype.OFF);//rumena
			END_IF
			ldDr1(ledChannel := 1);
			//ldDr2(ledChannel := 2);
			ldDr3(ledChannel := 3);
			axDR(calibParameters := JoystickGVL.calibration);
			
			JoystickGVL.xSpeed := axDr.xAxis;
			JoystickGVL.ySpeed := axDr.yAxis;
			JoystickGVL.zSpeed := axDr.zAxis;
			
			IF button = ButtonType.pressed AND JoystickGVL.speedScale = 1.0 AND JoystickGVL.intState = InternalState.override THEN
				JoystickGVL.speedScale := 0.5;
				ldDr1(ledChannel := 1, ledBlink := LEDtype.OFF);//rumena
				ldDr1(ledChannel := 1, ledBlink := LEDtype.Pulse, blinkInterval := T#1S);//rumena
			ELSIF button = ButtonType.pressed AND JoystickGVL.speedScale = 0.5 AND JoystickGVL.intState = InternalState.override THEN
				ldDr1(ledChannel := 1, ledBlink := LEDtype.OFF);//rumena
				ldDr1(ledChannel := 1, ledBlink := LEDtype.Pulse, blinkInterval := T#0.5S);//rumena
				JoystickGVL.speedScale := 1.0;
			ELSIF button = ButtonType.hold2s THEN
				//change internal state
				changeState := TRUE;
			ELSIF button = ButtonType.hold5s THEN
				initOp := TRUE;
				JoystickGVL.state := JoystickState.Calib;
				ldDr1(ledChannel := 1, ledBlink := LEDtype.OFF);//zelena
				//ldDr2(ledChannel := 2, ledBlink := LEDtype.OFF);//rumena
				ldDr3(ledChannel := 3, ledBlink := LEDtype.OFF);//rdeca
				prevStateCal := 0;
				calFB.reset();
				init := TRUE;
			END_IF
			
			IF changeState THEN
				changeState := FALSE;
				CASE JoystickGVL.intState OF
					InternalState.override:
						JoystickGVL.intState := InternalState.udpOnly;
						ControlGVL.status := ControlGVL.status AND 2#11111111111111111111111111111101;
						ControlGVL.status := ControlGVL.status OR 2#00000000000000000000000000000100;
						ldDr3(ledChannel := 3, ledBlink := LEDtype.OFF);
						ldDr3(ledChannel := 3, ledBlink := LEDtype.ON);
						ldDr1(ledChannel := 1, ledBlink := LEDtype.OFF);//rumena
						JoystickGVL.speedScale := 0.0;
						JoystickGVL.lastUpdate := TRUE;
					InternalState.passive:
						JoystickGVL.intState := InternalState.override;
						ControlGVL.status := ControlGVL.status OR 2#00000000000000000000000000000010;
						ldDr3(ledChannel := 3, ledBlink := LEDtype.OFF);
						ldDr3(ledChannel := 3, ledBlink := LEDtype.Pulse, blinkInterval := T#0.5S);
						JoystickGVL.speedScale := 0.5;
						ldDr1(ledChannel := 1, ledBlink := LEDtype.OFF);//rumena
						ldDr1(ledChannel := 1, ledBlink := LEDtype.Pulse, blinkInterval := T#1S);//rumena
					InternalState.udpOnly:
						JoystickGVL.intState := InternalState.passive;
						ControlGVL.status := ControlGVL.status AND 2#11111111111111111111111111111011;
						
						ldDr3(ledChannel := 3, ledBlink := LEDtype.OFF);
						//ldDr3(ledChannel := 3, ledBlink := LEDtype.ON);
						ldDr1(ledChannel := 1, ledBlink := LEDtype.OFF);//rumena
						ldDr1(ledChannel := 1, ledBlink := LEDtype.ON);//rumena
						
						JoystickGVL.speedScale := 0.0;
						JoystickGVL.lastUpdate := TRUE;
				END_CASE
			END_IF
			
			IF JoystickGVL.intState = InternalState.udpOnly THEN
				//Udp joystick stuff
				IF JoystickGVL.xSpeed > 0 THEN
					ControlGVL.status := ControlGVL.status OR 2#00000000000000000000000000001000;
				ELSIF JoystickGVL.xSpeed < 0 THEN
					ControlGVL.status := ControlGVL.status OR 2#00000000000000000000000000010000;
				ELSE
					ControlGVL.status := ControlGVL.status AND 2#11111111111111111111111111100111;
				END_IF
				IF JoystickGVL.ySpeed > 0 THEN
					ControlGVL.status := ControlGVL.status OR 2#00000000000000000000000000100000;
				ELSIF JoystickGVL.ySpeed < 0 THEN
					ControlGVL.status := ControlGVL.status OR 2#00000000000000000000000001000000;
				ELSE
					ControlGVL.status := ControlGVL.status AND 2#11111111111111111111111110011111;
				END_IF
				IF JoystickGVL.zSpeed > 0 THEN
					ControlGVL.status := ControlGVL.status OR 2#00000000000000000000000010000000;
				ELSIF JoystickGVL.zSpeed < 0 THEN
					ControlGVL.status := ControlGVL.status OR 2#00000000000000000000000100000000;
				ELSE
					ControlGVL.status := ControlGVL.status AND 2#11111111111111111111111001111111;
				END_IF
				IF button = ButtonType.pressed THEN
					ControlGVL.status := ControlGVL.status OR 2#00000000000000000000001000000000;
				ELSE
					ControlGVL.status := ControlGVL.status AND 2#11111111111111111111110111111111;
				END_IF
			END_IF
			
		
	END_CASE
END_IF

END_PROGRAM

// ---- POUs/Joystick/FBs/AXISdriver.TcPOU
FUNCTION_BLOCK AXISdriver
VAR_INPUT
	calibParameters : ST_Calibration_Parameters;
END_VAR
VAR_OUTPUT
	xAxis : LREAL := 0.0;
	yAxis : LREAL := 0.0;
	zAxis : LREAL := 0.0;
	
	xRawOut : INT := 0;
	yRawOut : INT := 0;
	zRawOut : INT := 0;
	
	xFilterOut : LREAL := 0.0;
	yFilterOut : LREAL := 0.0;
	zFilterOut : LREAL := 0.0;
END_VAR
VAR
	xRaw AT %I* : INT;
	yRaw AT %I* : INT;
	zRaw AT %I* : INT;
	
	xFilter : LREAL := 0.0;
	yFilter : LREAL := 0.0;
	zFilter : LREAL := 0.0;
END_VAR
VAR CONSTANT
	filter : LREAL := 0.1;
END_VAR

xRawOut := xRaw;
yRawOut := zRaw;
zRawOut := yRaw;

xFilter := xFilter * filter + (1 - filter) * INT_TO_LREAL(xRaw);
yFilter := yFilter * filter + (1 - filter) * INT_TO_LREAL(zRaw);
zFilter := zFilter * filter + (1 - filter) * INT_TO_LREAL(yRaw);

xFilterOut := xFilter;
yFilterOut := yFilter;
zFilterOut := zFilter;

IF JoystickGVL.state = JoystickState.Operational THEN
	IF (calibParameters.deadband[1] - ABS(xFilter - calibPArameters.zero[1])) > 0 THEN
		xAxis := 0.0;		
	ELSE
		xAxis := xFilter/(INT_TO_LREAL(calibParameters.maximums[1])-INT_TO_LREAL(calibParameters.zero[1]))+(-INT_TO_LREAL(calibParameters.zero[1])/(INT_TO_LREAL(calibParameters.maximums[1])-INT_TO_LREAL(calibParameters.zero[1])));
	END_IF
	
	IF (calibParameters.deadband[2] - ABS(yFilter - calibPArameters.zero[2])) > 0 THEN
		yAxis := 0.0;		
	ELSE
		yAxis := yFilter/(INT_TO_LREAL(calibParameters.maximums[2])-INT_TO_LREAL(calibParameters.zero[2]))+(-INT_TO_LREAL(calibParameters.zero[2])/(INT_TO_LREAL(calibParameters.maximums[2])-INT_TO_LREAL(calibParameters.zero[2])));
	END_IF
	
	IF (calibParameters.deadband[3] - ABS(zFilter - calibPArameters.zero[3])) > 0 THEN
		zAxis := 0.0;		
	ELSE
		zAxis := zFilter/(INT_TO_LREAL(calibParameters.maximums[3])-INT_TO_LREAL(calibParameters.zero[3]))+(-INT_TO_LREAL(calibParameters.zero[3])/(INT_TO_LREAL(calibParameters.maximums[3])-INT_TO_LREAL(calibParameters.zero[3])));
	END_IF

END_IF

END_FUNCTION_BLOCK

// ---- POUs/Joystick/FBs/BUTTONdriver.TcPOU
FUNCTION_BLOCK BUTTONdriver
VAR_INPUT
	buttonChannel : UINT := 1;
END_VAR
VAR_OUTPUT
END_VAR
VAR
	ch1 AT %I* : BOOL;
	ch2 AT %I* : BOOL;
	ch3 AT %I* : BOOL;
	ch4 AT %I* : BOOL;
	ch5 AT %I* : BOOL;
	ch6 AT %I* : BOOL;
	ch7 AT %I* : BOOL;
	ch8 AT %I* : BOOL;
	
	tmr1 : TON;
	currentValue : BOOL := FALSE;
	executed : BOOL := FALSE;
	
	state : ButtonType := ButtonType.notPressed;
END_VAR

CASE buttonChannel OF
	1:
		currentValue := ch1;
	2:
		currentValue := ch2;
	3:
		currentValue := ch3;
	4:
		currentValue := ch4;
	5:
		currentValue := ch5;
	6:
		currentValue := ch6;
	7:
		currentValue := ch7;
	8:
		currentValue := ch8;
END_CASE

IF currentValue AND NOT executed THEN
	tmr1(IN := TRUE, PT := T#10S);
	executed := TRUE;
ELSIF executed AND NOT currentValue AND (tmr1.ET < T#2S) THEN
	//momentary press
	tmr1(IN := FALSE);
	executed := FALSE;
	state := buttonType.pressed;
ELSIF executed AND NOT currentValue AND (tmr1.ET > T#2S) AND (tmr1.ET < T#5S) THEN
	//2S press
	tmr1(IN := FALSE);
	executed := FALSE;
	state := buttonType.hold2s;
ELSIF executed AND NOT currentValue AND (tmr1.ET > T#5S) THEN
	//5S press
	tmr1(IN := FALSE);
	executed := FALSE;
	state := buttonType.hold5s;
ELSIF executed AND tmr1.Q THEN
	//longer than 10S
	tmr1(IN := FALSE);
	executed := FALSE;
	state := buttonType.hold5s;
END_IF
tmr1();

METHOD getValue : BOOL
VAR_INPUT
END_VAR
VAR_OUTPUT
	stateOut : ButtonType;
END_VAR
stateOut := state;
state := ButtonType.notPressed;
getValue := TRUE;
END_METHOD

END_FUNCTION_BLOCK

// ---- POUs/Joystick/FBs/LEDdriver.TcPOU
FUNCTION_BLOCK LEDdriver
VAR_INPUT
	ledBlink : LEDtype;
	blinkInterval : TIME;
	
	ledChannel : UINT := 1;
END_VAR
VAR_OUTPUT
END_VAR
VAR
	ch1 AT %Q* : BOOL ;
	ch2 AT %Q* : BOOL ;
	ch3 AT %Q* : BOOL ;
	ch4 AT %Q* : BOOL ;
	ch5 AT %Q* : BOOL ;
	ch6 AT %Q* : BOOL ;
	ch7 AT %Q* : BOOL ;
	ch8 AT %Q* : BOOL ;
	
	ch1mode AT %Q* : BOOL;
	ch2mode AT %Q* : BOOL;
	ch3mode AT %Q* : BOOL;
	ch4mode AT %Q* : BOOL;
	ch5mode AT %Q* : BOOL;
	ch6mode AT %Q* : BOOL;
	ch7mode AT %Q* : BOOL;
	ch8mode AT %Q* : BOOL;
	
	tmr1 : TON;
	
	value : BOOL := FALSE;
	currentValue : BOOL := FALSE;
	executed : BOOL := FALSE;
END_VAR

CASE ledChannel OF
	1:
		currentValue := ch1;
	2:
		currentValue := ch2;
	3:
		currentValue := ch3;
	4:
		currentValue := ch4;
	5:
		currentValue := ch5;
	6:
		currentValue := ch6;
	7:
		currentValue := ch7;
	8:
		currentValue := ch8;
END_CASE

CASE ledBlink OF
	LEDtype.OFF:
		value := FALSE;
		executed := FALSE;
	LEDtype.ON:
		value := TRUE;
	LEDtype.BlinkOnce:
		IF currentValue AND tmr1.Q THEN
			value := FALSE;
			tmr1(IN := FALSE);
			executed := TRUE;
		ELSIF NOT executed THEN
			value := TRUE;
			tmr1(IN := TRUE, PT := T#0.5S);
		END_IF
	LEDtype.BlinkContinious:
		IF currentValue AND tmr1.Q THEN
			value := FALSE;
			tmr1(IN := FALSE);
			tmr1(IN := TRUE, PT := blinkInterval);
			executed := TRUE;
		ELSIF NOT currentValue AND tmr1.Q THEN
			value := TRUE;
			tmr1(IN := FALSE);
			tmr1(IN := TRUE, PT := blinkInterval);
		ELSIF NOT executed THEN
			executed := TRUE;
			tmr1(IN := TRUE, PT := T#0.01S);
		ELSE
			tmr1();
		END_IF
	LEDtype.Pulse:
		IF currentValue AND tmr1.Q THEN
			value := FALSE;
			tmr1(IN := FALSE);
			tmr1(IN := TRUE, PT := blinkInterval);
			executed := TRUE;
		ELSIF NOT currentValue AND tmr1.Q THEN
			value := TRUE;
			tmr1(IN := FALSE);
			tmr1(IN := TRUE, PT := T#0.01S);
		ELSIF NOT executed THEN
			executed := TRUE;
			tmr1(IN := TRUE, PT := T#0.01S);
		ELSE
			tmr1();
		END_IF
END_CASE

CASE ledChannel OF
	1:
		ch1mode := TRUE;
		ch1 := value;
	2:
		ch2mode := TRUE;
		ch2 := value;
	3:
		ch3mode := TRUE;
		ch3 := value;
	4:
		ch4mode := TRUE;
		ch4 := value;
	5:
		ch5mode := TRUE;
		ch5 := value;
	6:
		ch6mode := TRUE;
		ch6 := value;
	7:
		ch7mode := TRUE;
		ch7 := value;
	8:
		ch8mode := TRUE;
		ch8 := value;
	9:
		ch1mode := FALSE;
		ch2mode := FALSE;
		ch3mode := FALSE;
		ch4mode := FALSE;
		ch5mode := FALSE;
		ch6mode := FALSE;
		ch7mode := FALSE;
		ch8mode := FALSE;
END_CASE

END_FUNCTION_BLOCK

// ---- POUs/Joystick/FBs/CalibrationFB.TcPOU
FUNCTION_BLOCK CalibrationFB
VAR_INPUT
	buttonState : ButtonType := ButtonType.notPressed;
END_VAR
VAR_OUTPUT
	finished : BOOL := FALSE;
	stage1 : BOOL := TRUE;
	stage2 : BOOL := FALSE;
	stage3 : BOOL := FALSE;
	calibrationParams : ST_Calibration_Parameters;
	calLight : BOOL := FALSE;
END_VAR
VAR
	calParam : ST_Calibration_Parameters;
	maxDeadband : INT;
	
	zero : ARRAY [1..3] OF INT;
	zeroVals : ARRAY [1..1000] OF ARRAY [1..3] OF INT;
	zeroIterator : INT := 0;
	
	deadbandMax : ARRAY [1..3] OF INT := [-INT#32000,-INT#32000,-INT#32000];
	deadbandMin : ARRAY [1..3] OF INT := [INT#32000,INT#32000,INT#32000];
	
	MaxJs : ARRAY [1..3] OF INT := [-INT#32000,-INT#32000,-INT#32000];
	MinJs : ARRAY [1..3] OF INT := [INT#32000,INT#32000,INT#32000];
	
	axDr : AXISdriver;
END_VAR

axDr();
calLight := FALSE;
IF stage1 THEN
	//Zero
	zeroIterator := zeroIterator + 1;
	zeroVals[zeroIterator][1] := LREAL_TO_INT(axDr.xFilterOut);
	zeroVals[zeroIterator][2] := LREAL_TO_INT(axDr.yFilterOut);
	zeroVals[zeroIterator][3] := LREAL_TO_INT(axDr.zFilterOut);
	IF zeroIterator > 999 THEN
		zero[1] := (zeroVals[300][1] + zeroVals[400][1] + zeroVals[500][1] + zeroVals[600][1])/4;
		zero[2] := (zeroVals[300][2] + zeroVals[400][2] + zeroVals[500][2] + zeroVals[600][2])/4;
		zero[3] := (zeroVals[300][3] + zeroVals[400][3] + zeroVals[500][3] + zeroVals[600][3])/4;
		calParam.zero := zero;
		zeroIterator := 0;
		stage1 := FALSE;
		stage2 := TRUE;
	END_IF
	
ELSIF stage2 THEN
	//deadband
	IF LREAL_TO_INT(axDr.xFilterOut) > deadbandMax[1] THEN
		deadbandMax[1] := LREAL_TO_INT(axDr.xFilterOut);
		calLight := TRUE;
	END_IF
	IF LREAL_TO_INT(axDr.yFilterOut) > deadbandMax[2] THEN
		deadbandMax[2] := LREAL_TO_INT(axDr.yFilterOut);
		calLight := TRUE;
	END_IF
	IF LREAL_TO_INT(axDr.zFilterOut) > deadbandMax[3] THEN
		deadbandMax[3] := LREAL_TO_INT(axDr.zFilterOut);
		calLight := TRUE;
	END_IF
	IF LREAL_TO_INT(axDr.xFilterOut) < deadbandMin[1] THEN
		deadbandMin[1] := LREAL_TO_INT(axDr.xFilterOut);
		calLight := TRUE;
	END_IF
	IF LREAL_TO_INT(axDr.yFilterOut) < deadbandMin[2] THEN
		deadbandMin[2] := LREAL_TO_INT(axDr.yFilterOut);
		calLight := TRUE;
	END_IF
	IF LREAL_TO_INT(axDr.zFilterOut) < deadbandMin[3] THEN
		deadbandMin[3] := LREAL_TO_INT(axDr.zFilterOut);
		calLight := TRUE;
	END_IF
	IF buttonState = buttonType.pressed THEN
		stage2 := FALSE;
		stage3 := TRUE;
		calParam.deadband[1] := (deadbandMax[1] - deadbandMin[1])/2 + 250;
		calParam.deadband[2] := (deadbandMax[2] - deadbandMin[2])/2 + 250;
		calParam.deadband[3] := (deadbandMax[3] - deadbandMin[3])/2 + 250;
	END_IF
ELSIF stage3 THEN
	//minmax
	IF LREAL_TO_INT(axDr.xFilterOut) > MaxJs[1] THEN
		MaxJs[1] := LREAL_TO_INT(axDr.xFilterOut);
		calLight := TRUE;
	END_IF
	IF LREAL_TO_INT(axDr.yFilterOut) > MaxJs[2] THEN
		MaxJs[2] := LREAL_TO_INT(axDr.yFilterOut);
		calLight := TRUE;
	END_IF
	IF LREAL_TO_INT(axDr.zFilterOut) > MaxJs[3] THEN
		MaxJs[3] := LREAL_TO_INT(axDr.zFilterOut);
		calLight := TRUE;
	END_IF
	IF LREAL_TO_INT(axDr.xFilterOut) < MinJs[1] THEN
		MinJs[1] := LREAL_TO_INT(axDr.xFilterOut);
		calLight := TRUE;
	END_IF
	IF LREAL_TO_INT(axDr.yFilterOut) < MinJs[2] THEN
		MinJs[2] := LREAL_TO_INT(axDr.yFilterOut);
		calLight := TRUE;
	END_IF
	IF LREAL_TO_INT(axDr.zFilterOut) < MinJs[3] THEN
		MinJs[3] := LREAL_TO_INT(axDr.zFilterOut);
		calLight := TRUE;
	END_IF
	IF buttonState = buttonType.pressed THEN
		stage2 := FALSE;
		stage3 := FALSE;
		calParam.maximums[1] := MaxJs[1];
		calParam.maximums[2] := MaxJs[2];
		calParam.maximums[3] := MaxJs[3];
		calParam.minimums[1] := MinJs[1];
		calParam.minimums[2] := MinJs[2];
		calParam.minimums[3] := MinJs[3];
		calParam.calibrated := TRUE;
	END_IF
ELSE
	stage1 := TRUE;
	finished := TRUE;
	calibrationParams := calParam;
END_IF

METHOD reset : BOOL
VAR_INPUT
END_VAR
finished := FALSE;
stage1 := TRUE;
stage2 := FALSE;
stage3 := FALSE;
calLight := FALSE;

zeroIterator := 0;

deadbandMax[1] := -INT#32000;
deadbandMax[2] := -INT#32000;
deadbandMax[3] := -INT#32000;

deadbandMin[1] := INT#32000;
deadbandMin[2] := INT#32000;
deadbandMin[3] := INT#32000;
	
MaxJs[1] := -INT#32000;
MaxJs[2] := -INT#32000;
MaxJs[3] := -INT#32000;

MinJs[1] := INT#32000;
MinJs[2] := INT#32000;
MinJs[3] := INT#32000;

reset := TRUE;
END_METHOD

END_FUNCTION_BLOCK

// ---- POUs/Sensors/SensorsMain.TcPOU
PROGRAM SensorsMain
VAR
	
	angleDir : LREAL;
	

	
	sensor_D AT %Q* : BOOL;
	sensor_E AT %Q* : BOOL;
	sensor_F AT %Q* : BOOL;
	
	
	
	
	en_sensor_D AT %Q* : BOOL ;
	en_sensor_E AT %Q* : BOOL ;
	en_sensor_F AT %Q* : BOOL ;


	sensor1_UO1 AT %I* : BOOL;
	sensor1_UO2 AT %I* : BOOL;
	sensor1_UO3 AT %I* : BOOL;
	
	sensor2_UO1 AT %I* : BOOL;
	sensor2_UO2 AT %I* : BOOL;
	sensor2_UO3 AT %I* : BOOL;
	
	tmr1 : TON; //program period
	new_direction : INT := 0; //new direction based on velocity direction
	direction : ARRAY [0..8] OF INT := [0,0,0,0,0,0,0,0,0]; //stock last new directions
	lastChange : LREAL := 0; //prevent to change fields too quickly 
	Index : INT := 0;
	maxVal : INT := -1;
	
	
	
	
	
END_VAR

VAR CONSTANT
	PI_8 : LREAL := 0.39269908169872414;
	VMAX : LREAL := 1.2;
	VTHMAX : LREAL := 0.5;
	TPROG : LREAL := 0.001;
	TWAIT : LREAL := 0.2;
 	

END_VAR

//Compute acctual direction of the mobile platform
IF(ABS(ControlGVL.forwardReverse)<0.04) THEN
	IF(ControlGVL.leftRight>0.04) THEN
		new_direction := DirPlatform.PLUS_Y;
	ELSIF(ControlGVL.leftRight<-0.04) THEN
		new_direction := DirPlatform.MINUS_Y;
	ELSE
		new_direction := DirPlatform.PLUS_X; //assume default field is Plus X
	END_IF

ELSE
	angleDir := ATAN(-ControlGVL.leftRight/ControlGVL.forwardReverse);
	IF(ControlGVL.forwardReverse<0) THEN
		angleDir := angleDir + 3.141592;
	END_IF

	IF((angleDir>=PI_8)AND(angleDir<3*PI_8)) THEN
		new_direction := DirPlatform.PLUS_X_MINUS_Y;
	ELSIF((angleDir>=3*PI_8)AND(angleDir<5*PI_8)) THEN
		new_direction := DirPlatform.MINUS_Y;
	ELSIF((angleDir>=5*PI_8)AND(angleDir<7*PI_8)) THEN
		new_direction := DirPlatform.MINUS_X_MINUS_Y;
	ELSIF((angleDir>=7*PI_8)AND(angleDir<9*PI_8)) THEN
		new_direction := DirPlatform.MINUS_X;
	ELSIF((angleDir>=9*PI_8)AND(angleDir<11*PI_8)) THEN
		new_direction := DirPlatform.MINUS_X_PLUS_Y;
	ELSIF(((angleDir>=11*PI_8)AND(angleDir<12*PI_8))OR((angleDir>=-4*PI_8)AND(angleDir<-3*PI_8))) THEN
		new_direction := DirPlatform.PLUS_Y;
	ELSIF((angleDir>=-3*PI_8)AND(angleDir<-1*PI_8)) THEN
		new_direction := DirPlatform.PLUS_X_PLUS_Y;
	ELSE
		new_direction := DirPlatform.PLUS_X;
	END_IF
END_IF


//prevent to change too often the set of fields
lastChange := lastChange + TPROG;
//store the new_direction of the cycle
direction[new_direction] := direction[new_direction] +1;
IF((lastChange>TWAIT)) THEN //possibly change only each TWAIT seconds
	
	maxVal := -1;
	FOR Index := 0 TO 8 DO //find the direction most asked
		IF direction[Index] > maxVal THEN
			maxVal := direction[Index];
			new_direction := Index;
		END_IF
		//reset variable for another cycle
  		direction[Index] := 0;
	END_FOR

	SensorsGVL.platformDir := new_direction; //update the fields
	lastChange := 0;
END_IF






//emable writting output
en_sensor_D := TRUE;
en_sensor_E := TRUE;
en_sensor_F := TRUE;



//Update fields on sensors
sensor_D := (SensorsGVL.platformDir / 4)>0;
sensor_E := ((SensorsGVL.platformDir MOD 4)/2)>0;
sensor_F := (SensorsGVL.platformDir MOD 2) >0;




//Adapt maximum speed if obstacles
IF (sensor1_UO1 OR sensor2_UO1) THEN
	ControlGVL.currentVelMax := 0;
	ControlGVL.currentThVelMax :=0;
ELSIF (sensor1_UO2 OR sensor2_UO2) THEN
	ControlGVL.currentVelMax := VMAX/4;
	ControlGVL.currentThVelMax :=VTHMAX;
ELSIF (sensor1_UO3 OR sensor2_UO3) THEN
	ControlGVL.currentVelMax := VMAX/2;
	ControlGVL.currentThVelMax :=VTHMAX;
ELSE
	ControlGVL.currentVelMax := VMAX;
	ControlGVL.currentThVelMax :=VTHMAX;
END_IF

ControlGVL.currentVelMax := VMAX/2;
ControlGVL.currentThVelMax :=VTHMAX;

END_PROGRAM
